# B&R Automation Studio project Tmp_Explorer_V1 (part 2)

#### Main.st - not listed in the package file held
```iecst
// ----------------------------------------------------------------------------------------
//	Function:	mappView explorer
//  Version:	1.08
//	Changed:	03.05.2021
// ----------------------------------------------------------------------------------------

PROGRAM _INIT
	// ----------------------------------------------------------------------------------------
	// Copy pre-configured devices into list
	brsmemcpy(ADR(EXPL.PAR[0].device_list), ADR(EXPL_DEVICE_LIST), SIZEOF(EXPL_DEVICE_LIST));
	brsmemcpy(ADR(EXPL.PAR[1].device_list), ADR(EXPL_DEVICE_LIST), SIZEOF(EXPL_DEVICE_LIST));
	brsstrcpy(ADR(EXPL.PAR[0].device_active), ADR(EXPL.PAR[0].device_list[0]));
	brsstrcpy(ADR(EXPL.PAR[1].device_active), ADR(EXPL.PAR[1].device_list[0]));

	// ----------------------------------------------------------------------------------------
	// Allocate memory for file upload and download
	AsMemPartCreate_0.enable	:= TRUE;
	AsMemPartCreate_0.len		:= EXPL_UPLOAD_DOWNLOAD_SIZE;
	AsMemPartCreate_0();
	IF AsMemPartCreate_0.status <> 0 THEN
		step := CreateError(ERR_MEM_ALLOC, side, step, 'file upload and download alloc failed', ADR(EXPL));
	ELSE
		AsMemPartAllocClear_0.enable	:= TRUE;
		AsMemPartAllocClear_0.ident		:= AsMemPartCreate_0.ident;
		AsMemPartAllocClear_0.len		:= EXPL_UPLOAD_DOWNLOAD_SIZE;
		AsMemPartAllocClear_0();
		IF AsMemPartCreate_0.status <> 0 THEN
			step := CreateError(ERR_MEM_ALLOC, side, step, 'file upload and download clear failed', ADR(EXPL));
		END_IF
	END_IF

	// ----------------------------------------------------------------------------------------
	// Generate HTML messages for web upload
	upload_response[0]	:= '<html><body><form action="/uploadA.html" name="form_upload" method="post" enctype="multipart/form-data" >
	<label for="file-upload" style="font-weight:bold;font-family: sans-serif;font-size:16px;padding:10px 10px;10px;10px;" class="custom-file-upload">Upload</label>
	<input type="file" id="file-upload" style="display:none;" onchange="form.submit()" name="file_selected" content-type="application/octet-stream" />
	</form><body></html> ';
	WebServiceUpload[0].pServiceName := ADR('uploadA.html');
	upload_response[1]	:= '<html><body><form action="/uploadB.html" name="form_upload" method="post" enctype="multipart/form-data" >
	<label for="file-upload" style="font-weight:bold;font-family: sans-serif;font-size:16px;padding:10px 10px;10px;10px;" class="custom-file-upload">Upload</label>
	<input type="file" id="file-upload" style="display:none;" onchange="form.submit()" name="file_selected" content-type="application/octet-stream" />
	</form><body></html> ';
	WebServiceUpload[1].pServiceName := ADR('uploadB.html');

	// ----------------------------------------------------------------------------------------
	// Connect to user device for temporary files used with download all
	REPEAT
		DevLink_0.enable := 1;
		DevLink_0.pDevice := ADR('TMP_USER');
		DevLink_0.pParam := ADR('/DEVICE=F:');
		DevLink_0;
		UNTIL DevLink_0.status <> ERR_FUB_BUSY
	END_REPEAT;
END_PROGRAM

PROGRAM _CYCLIC
	// ----------------------------------------------------------------------------------------
	// Web service driver for file upload
	WebServiceUpload[side].enable 			:= TRUE;
	WebServiceUpload[side].option 			:= httpOPTION_HTTP_11 + httpOPTION_SERVICE_TYPE_NAME;
	WebServiceUpload[side].pRequestData  	:= AsMemPartAllocClear_0.mem;
	WebServiceUpload[side].requestDataSize 	:= EXPL_UPLOAD_DOWNLOAD_SIZE;
	WebServiceUpload[side].pResponseData 	:= ADR(upload_response[side]);
	WebServiceUpload[side].responseDataLen 	:= brsstrlen(ADR(upload_response[side]));
	WebServiceUpload[side]();

	// Reset send command
	IF(WebServiceUpload[side].send = TRUE)  THEN
		WebServiceUpload[side].send := FALSE;
	// Send response when page is loaded or data is posted
	ELSIF(WebServiceUpload[side].status = ERR_OK AND WebServiceUpload[side].send = FALSE) THEN
		WebServiceUpload[side].send := TRUE;
	// New upload data arrived
	ELSIF(WebServiceUpload[side].send = FALSE AND WebServiceUpload[side].requestDataLen > 0 AND EXPL.CMD[side].upload = FALSE) THEN
		// Add delay so that upload can finish
		upload_delay.PT := WebServiceUpload[side].requestDataLen/100000*5;
		upload_delay.IN := TRUE;
		upload_delay();
	END_IF
	// Check new uploaded data
	IF(upload_delay.Q AND EXPL.CMD[side].upload = FALSE) THEN
		upload_delay.IN := FALSE;
		upload_delay();
		EXPL.CMD[side].upload := TRUE;
	END_IF

	// ------------------------------------------------------------------------------------------------
	// Set switches for HMI, these buttons are enabled if there is at least one file or directory
	IF(EXPL.DAT[side].item_num > 0) THEN
		EXPL.VIS[side].enable_button_set_1 := TRUE;
	ELSE
		EXPL.VIS[side].enable_button_set_1 := FALSE;
	END_IF

	// ------------------------------------------------------------------------------------------------
	// Generate device name list for drop down box
	brsmemset(ADR(EXPL.VIS[side].device_list), 0, SIZEOF(EXPL.VIS[side].device_list));
	FOR lx := 0 TO SIZEOF(EXPL.VIS[side].device_list)/SIZEOF(EXPL.VIS[side].device_list[0]) - 1 DO
		IF (EXPL.PAR[side].device_list[lx] <> '') THEN
			String2DataProvider(ADR(EXPL.PAR[side].device_list[lx]), ADR(EXPL.VIS[side].device_list[lx]));
		END_IF
	END_FOR;

	// ------------------------------------------------------------------------------------------------
	// Handle double click for directory change and file view
	IF(EXPL.VIS[side].double_click_event > 0) THEN
		double_click_timer.PT := 50;
		double_click_timer.IN := TRUE;
		double_click_timer();
		IF(EXPL.VIS[side].double_click_event > 1) THEN
			double_click_timer.IN := FALSE;
			double_click_timer();
			EXPL.VIS[side].double_click_event := 0;
			IF(brsmemcmp(ADR(EXPL.DAT[side].item_list[EXPL.VIS[side].item_selected]), ADR('(DIR)'), 5) = 0 OR EXPL.DAT[side].item_list[EXPL.VIS[side].item_selected] = '..') THEN
				EXPL.CMD[side].dir_change := TRUE;
			ELSE
				EXPL.CMD[side].view_file := TRUE;
			END_IF
		END_IF
	END_IF
	IF(double_click_timer.Q) THEN
		double_click_timer.IN := FALSE;
		double_click_timer();
		IF(EXPL.VIS[side].double_click_event > 0) THEN
			EXPL.VIS[side].double_click_event := EXPL.VIS[side].double_click_event - 1;
		END_IF
	END_IF

	//--------------------------------------------------------------------------------------------------
	// Check if parameters are valid
	IF (EXPL.PAR[side].device_active = '') THEN
		step := CreateError(ERR_DEVICE_UNDEFINED, side, step, 'device is not defined', ADR(EXPL));
		RETURN;
	END_IF
	IF (brsstrlen(ADR(EXPL.PAR[side].dir_path)) >= EXPL_DIR_PATH_LENGTH) THEN
		step := CreateError(ERR_PATH_CRITICAL, side, step, 'directory path critical error', ADR(EXPL));
		RETURN;
	END_IF

	// ------------------------------------------------------------------------------------------------
	// Track filter change
	IF (FILTER_AUTO_REFRESH AND brsstrcmp(ADR(old_filter[side]), ADR(EXPL.PAR[side].item_filter)) <> 0) THEN
		brsstrcpy(ADR(old_filter[side]), ADR(EXPL.PAR[side].item_filter));
		EXPL.CMD[side].refresh	:= TRUE;
	END_IF

	// ------------------------------------------------------------------------------------------------
	// Track device name change
	IF(device_active_old[side] <> EXPL.PAR[side].device_active) THEN
		EXPL.PAR[side].dir_path := '';
		EXPL.CMD[side].refresh	:= TRUE;
	END_IF
	device_active_old[side] := EXPL.PAR[side].device_active;

	// ------------------------------------------------------------------------------------------------
	// Stop here if no command is set
	IF (EXPL.CMD[side].refresh = FALSE AND EXPL.CMD[side].dir_change = FALSE AND EXPL.CMD[side].dir_create = FALSE AND EXPL.CMD[side].copy = FALSE AND EXPL.CMD[side].copy_all = FALSE AND EXPL.CMD[side].delete = FALSE AND EXPL.CMD[side].rename = FALSE AND EXPL.CMD[side].view_file = FALSE AND EXPL.CMD[side].download = FALSE AND EXPL.CMD[side].upload = FALSE) THEN
		// --------------------------------------------------------------------------------------------
		// Show current state
		EXPL.status_text := 'Waiting...';
		// --------------------------------------------------------------------------------------------
		// If selection is out of range set it to maximum
		IF ((EXPL.VIS[side].item_selected > EXPL.DAT[side].item_num - 1) AND (EXPL.DAT[side].item_num <> 0)) THEN
			EXPL.VIS[side].item_selected := EXPL.DAT[side].item_num - 1;
		END_IF
		side := NOT side;
		// Enable buttons when command is active
		EXPL.VIS[0].enable_button_set_2 := TRUE;
		EXPL.VIS[1].enable_button_set_2 := TRUE;
		// Reset busy status
		IF(EXPL.ERR.state = 0) THEN
			EXPL.status_no := 0;
		END_IF
		RETURN;
	END_IF

	// Disable buttons when command is active
	EXPL.VIS[0].enable_button_set_1 := FALSE;
	EXPL.VIS[1].enable_button_set_1 := FALSE;
	EXPL.VIS[0].enable_button_set_2 := FALSE;
	EXPL.VIS[1].enable_button_set_2 := FALSE;

	// Clear errors on new command
	brsmemset(ADR(EXPL.ERR), 0, SIZEOF(EXPL.ERR));

	//**************************************************************************************************
	// Cyclic Part
	//**************************************************************************************************
	CASE step OF
		//**********************************************************************************************
		// Wait for command
		//**********************************************************************************************
		EXP_WAIT:
			// ----------------------------------------------------------------------------------------
			// Refresh direcrory information
			IF (EXPL.CMD[side].refresh = TRUE) THEN
				step := EXP_READ_DIR;
			END_IF
			// ----------------------------------------------------------------------------------------
			// Change active directory
			IF (EXPL.CMD[side].dir_change = TRUE) THEN
				// ------------------------------------------------------------------------------------
				// Check if directory name is empty
				IF (EXPL.DAT[side].item_list[EXPL.VIS[side].item_selected] = '') THEN
					step := CreateError(ERR_EMPTY_ITEM, side, step, 'directory name is empty', ADR(EXPL));
				// Check if directory name is valid
				ELSIF((brsmemcmp(ADR(EXPL.DAT[side].item_list[EXPL.VIS[side].item_selected]), ADR('(DIR)'), 5) <> 0) AND (EXPL.DAT[side].item_list[EXPL.VIS[side].item_selected] <> '..'))  THEN
					step := CreateError(ERR_INVALID_ITEM_NAME, side, step, 'this is not a valid directory name', ADR(EXPL));
				// Check if new directory name fits into string
				ELSIF(brsstrlen(ADR(EXPL.DAT[side].item_list[EXPL.VIS[side].item_selected])) - 5 + brsstrlen(ADR(EXPL.PAR[side].dir_path)) + 1 >= EXPL_DIR_PATH_LENGTH) THEN
					step := CreateError(ERR_PATH_EXCEEDS_MAX, side, step, 'directory path exceeds maximum length', ADR(EXPL));
				ELSE
					step := EXP_DIR_CHANGE;
				END_IF
			END_IF
			// ----------------------------------------------------------------------------------------
			// Create a new directory
			IF (EXPL.CMD[side].dir_create = TRUE) THEN
				// ------------------------------------------------------------------------------------
				// Check if new directory name is empty
				IF (EXPL.PAR[side].new_name = '') THEN
					step := CreateError(ERR_EMPTY_ITEM, side, step, 'directory name is empty', ADR(EXPL));
				// Check if new directory name fits into path string
				ELSIF(brsstrlen(ADR(EXPL.PAR[side].new_name)) + brsstrlen(ADR(EXPL.PAR[side].dir_path)) + 1 >= EXPL_DIR_PATH_LENGTH) THEN
					step := CreateError(ERR_PATH_EXCEEDS_MAX, side, step, 'directory path name exceeds maximum length', ADR(EXPL));
				// Check if new directory name fits into directory name string
				ELSIF(brsstrlen(ADR(EXPL.PAR[side].new_name)) + 5 >= EXPL_ITEM_LENGTH) THEN
					step := CreateError(ERR_DIR_EXCEEDS_MAX, side, step, 'directory name exceeds maximum length', ADR(EXPL));
				ELSE
					step := EXP_DIR_CREATE;
				END_IF
			END_IF
			// ----------------------------------------------------------------------------------------
			// Copy one file
			IF (EXPL.CMD[side].copy = TRUE) THEN
				// ------------------------------------------------------------------------------------
				// Make sure that user chooses a valid item
				IF (EXPL.DAT[side].item_list[EXPL.VIS[side].item_selected] = '..') THEN
					step := CreateError(ERR_INVALID_ITEM_NAME, side, step, 'this is not a valid item name', ADR(EXPL));
				ELSE
					item_name := EXPL.DAT[side].item_list[EXPL.VIS[side].item_selected];
					step := EXP_OVERWRITE_1;
				END_IF
			END_IF
			// ----------------------------------------------------------------------------------------
			// Copy all files and folders in this directory
			IF (EXPL.CMD[side].copy_all = TRUE) THEN
				step := EXP_COPY_ALL;
			END_IF
			// ----------------------------------------------------------------------------------------
			// View selected file
			IF (EXPL.CMD[side].view_file = TRUE) THEN
				step := EXP_FILE_VIEW;
			END_IF
			// ----------------------------------------------------------------------------------------
			// Download selected file or directory
			IF (EXPL.CMD[side].download = TRUE) THEN
				EXPL.VIS[side].download_file_url := '';
				item_name := EXPL.DAT[side].item_list[EXPL.VIS[side].item_selected];
				// Make sure selected entry is valid
				IF(brsmemcmp(ADR(item_name), ADR('..'), 2) <> 0) THEN
					// Check if selected item is a single file
					IF(brsmemcmp(ADR(item_name), ADR('(DIR)'), 5) <> 0) THEN
						device_active := EXPL.PAR[side].device_active;
						dir_path := EXPL.PAR[side].dir_path;
						step := EXP_FILE_DOWNLOAD;
					// Selected item is a directory
					ELSE
						ReplaceString(ADR(item_name), ADR('(DIR)'), ADR(''), TRUE);
						step := EXP_FILE_DOWNLOAD_DIR;
					END_IF
				ELSE
					step := CreateError(ERR_DIR_DOWNLOAD_INVALID, side, step, 'item is not a valid directory', ADR(EXPL));
				END_IF
			END_IF
			// ----------------------------------------------------------------------------------------
			// Upload a new file
			IF (EXPL.CMD[side].upload = TRUE) THEN
				step := EXP_FILE_UPLOAD;
			END_IF
			// ----------------------------------------------------------------------------------------
			// Delete the selected file
			IF (EXPL.CMD[side].delete = 1) THEN
				// Check if directory name is empty
				IF (EXPL.DAT[side].item_list[EXPL.VIS[side].item_selected] = '')	THEN
					step := CreateError(ERR_EMPTY_ITEM, side, step, 'item name is empty', ADR(EXPL));
					// Check if new directory name fits into string
				ELSIF(brsstrlen(ADR(EXPL.DAT[side].item_list[EXPL.VIS[side].item_selected])) + brsstrlen(ADR(EXPL.PAR[side].dir_path)) + 1 >= EXPL_DIR_PATH_LENGTH + EXPL_ITEM_LENGTH) THEN
					step := CreateError(ERR_PATH_EXCEEDS_MAX, side, step, 'directory path exceeds maximum length', ADR(EXPL));
					// Make sure that a valid item was selected
				ELSIF(EXPL.DAT[side].item_list[EXPL.VIS[side].item_selected] = '..') THEN
					step := CreateError(ERR_INVALID_ITEM_NAME, side, step, 'this is not a valid item name', ADR(EXPL));
					// Delete a directory
				ELSIF(brsmemcmp(ADR(EXPL.DAT[side].item_list[EXPL.VIS[side].item_selected]), ADR('(DIR)'), 5) = 0)	THEN
					item_name := EXPL.DAT[side].item_list[EXPL.VIS[side].item_selected];
					step := EXP_DIR_DELETE;
				// Delete a file
				ELSE
					item_name := EXPL.DAT[side].item_list[EXPL.VIS[side].item_selected];
					step := EXP_FILE_DELETE;
				END_IF
			END_IF
			// ----------------------------------------------------------------------------------------
			// Rename file or directory
			IF (EXPL.CMD[side].rename = TRUE) THEN
				// ------------------------------------------------------------------------------------
				// Check if new directory name is empty
				IF (EXPL.PAR[side].new_name = '') THEN
					step := CreateError(ERR_EMPTY_ITEM, side, step, 'new name is empty', ADR(EXPL));
				// Make sure that a valid item was selected
				ELSIF (EXPL.DAT[side].item_list[EXPL.VIS[side].item_selected] = '..') THEN
					step := CreateError(ERR_INVALID_ITEM_NAME, side, step, 'this is not a valid item name', ADR(EXPL));
				// Rename a directory
				ELSIF(brsmemcmp(ADR(EXPL.DAT[side].item_list[EXPL.VIS[side].item_selected]), ADR('(DIR)'), 5) = 0)	THEN
					step := EXP_DIR_RENAME;
				// Rename a file
				ELSE
					step := EXP_FILE_RENAME;
				END_IF
			END_IF

			// Set status
			EXPL.status_no := ERR_FUB_BUSY;

		//**********************************************************************************************
		// Read directory information
		//**********************************************************************************************
		EXP_READ_DIR:
			// Show current state
			animation := animation := WorkingStatus(ADR(EXPL), ADR('reading directory...'), animation);
			// ----------------------------------------------------------------------------------------
			// Clear all entrys
			brsmemset(ADR(EXPL.DAT[side]), 0, SIZEOF(EXPL.DAT[side]));
			EXPL.VIS[side].item_selected := 0;
			EXPL.DAT[side].item_num := 0;
			// ----------------------------------------------------------------------------------------
			// Add .. for directory up
			IF(EXPL.PAR[side].dir_path <> '/' AND EXPL.PAR[side].dir_path <> '') THEN
				EXPL.DAT[side].item_list[0] := '..';
				EXPL.DAT[side].item_num := 1;
			END_IF
			// ----------------------------------------------------------------------------------------
			// Set parameters and get device dir
			DInfo.enable 	:= TRUE;
			DInfo.pDevice	:= ADR(EXPL.PAR[side].device_active);
			DInfo.pPath 	:= ADR(EXPL.PAR[side].dir_path);
			DInfo();

			// ----------------------------------------------------------------------------------------
			// OK
			IF (DInfo.status = OK) THEN
				step := EXP_READ_DIR_1;
			// ----------------------------------------------------------------------------------------
			// Device is not available
			ELSIF (DInfo.status = fiERR_FILE_DEVICE) THEN
			 	EXPL.DAT[side].item_list[0] := 'not connected';
				step := CreateError(DInfo.status, side, step, 'not connected', ADR(EXPL));
			// ----------------------------------------------------------------------------------------
			// Device is not available
			ELSIF (DInfo.status = fiERR_DEVICE_MANAGER) THEN
				EXPL.DAT[side].item_list[0] := 'not connected';
				step := CreateError(DInfo.status, side, step, 'check device name and path', ADR(EXPL));
			// Error
			ELSIF (DInfo.status <> ERR_FUB_BUSY) THEN
				step := CreateError(DInfo.status, side, step, 'error dir info', ADR(EXPL));
			END_IF
		//**********************************************************************************************
		// Open directory
		//**********************************************************************************************
		EXP_READ_DIR_1:
			// Add current directory
			IF(EXPL.PAR[side].dir_path = '') THEN
				EXPL.PAR[side].dir_path := '/';
			END_IF
			DOpen.enable 	:= TRUE;
			DOpen.pDevice	:= ADR(EXPL.PAR[side].device_active);
			DOpen.pName 	:= ADR(EXPL.PAR[side].dir_path);
			DOpen();

			// ----------------------------------------------------------------------------------------
			// OK
			IF (DOpen.status = OK) THEN
				has_oversized_items := FALSE;
				step := EXP_READ_DIR_2;
			// Error
			ELSIF (DOpen.status <> ERR_FUB_BUSY) THEN
				step := CreateError(DOpen.status, side, step, 'error dir open', ADR(EXPL));
			END_IF;
		//**********************************************************************************************
		// Read file directory information
		//**********************************************************************************************
	 	EXP_READ_DIR_2:
			DRead.enable 	:= TRUE;
			DRead.ident		:= DOpen.ident;
			DRead.pData 	:= ADR(lDirReadData);
			DRead.data_len 	:= SIZEOF(lDirReadData);
			DRead();

			// ----------------------------------------------------------------------------------------
			// OK
			IF (DRead.status = OK) THEN
				// ------------------------------------------------------------------------------------
				// Verify that we still have space in list
				IF (EXPL.DAT[side].item_num < SIZEOF(EXPL.DAT[side].item_list)/SIZEOF(EXPL.DAT[side].item_list[0])) THEN
					// --------------------------------------------------------------------------------
					// Make sure file name contains filter
					IF (brsstrlen(ADR(EXPL.PAR[side].item_filter)) = 0 OR IsInstr(ADR(lDirReadData.Filename), ADR(EXPL.PAR[side].item_filter))) THEN
						brsmemset(ADR(tmp_str1), 0, SIZEOF(tmp_str1));
						// ----------------------------------------------------------------------------
						// Read file information
						IF (lDirReadData.Mode = fiFILE) THEN
							IF (brsstrlen(ADR(lDirReadData.Filename)) < EXPL_ITEM_LENGTH) THEN
								brsstrcpy(ADR(tmp_str1), ADR(lDirReadData.Filename));
								// --------------------------------------------------------------------
								// Generate file size
								IF (lDirReadData.Filelength > 1048576) THEN
									brsitoa(lDirReadData.Filelength/1048576, ADR(tmp_str2));
									brsstrcat(ADR(tmp_str2), ADR('M'));
								ELSIF (lDirReadData.Filelength > 1024) THEN
									brsitoa(lDirReadData.Filelength/1024, ADR(tmp_str2));
									brsstrcat(ADR(tmp_str2), ADR('K'));
								ELSE
									brsitoa(lDirReadData.Filelength, ADR(tmp_str2));
								END_IF
								InsertRecName(ADR(EXPL), tmp_str1, tmp_str2, side);
								EXPL.DAT[side].item_num := EXPL.DAT[side].item_num + 1;
							ELSE
								has_oversized_items := TRUE;
							END_IF
						// ----------------------------------------------------------------------------
						// Read directory information
						ELSIF (brsstrcmp(ADR(lDirReadData.Filename), ADR('.')) <> 0 AND brsstrcmp(ADR(lDirReadData.Filename), ADR('..')) <> 0 AND brsstrcmp(ADR(lDirReadData.Filename), ADR('System Volume Information')) <> 0) THEN
							IF (brsstrlen(ADR(lDirReadData.Filename)) < EXPL_ITEM_LENGTH-5) THEN
								// Copy directory name
								tmp_str1 := '(DIR)';
								brsstrcat(ADR(tmp_str1), ADR(lDirReadData.Filename));
								InsertRecName(ADR(EXPL), tmp_str1, '', side);
								EXPL.DAT[side].item_num := EXPL.DAT[side].item_num + 1;
							ELSE
								has_oversized_items := TRUE;
							END_IF
						END_IF
					END_IF
				ELSE
					step := CreateError(ERR_MAX_FILES_REACHED, side, step, 'maximum number of files reached', ADR(EXPL));
				END_IF
			// Last entry reached
			ELSIF (DRead.status = fiERR_NO_MORE_ENTRIES) THEN
				step := EXP_READ_DIR_3;
			// Error
			ELSIF (DRead.status <> ERR_FUB_BUSY) THEN
				step := CreateError(DRead.status, side, step, 'error dir read', ADR(EXPL));
			END_IF
		//**********************************************************************************************
		// Close directory information
		//**********************************************************************************************
		EXP_READ_DIR_3:
			DClose.enable 	:= TRUE;
			DClose.ident	:= DOpen.ident;
			DClose();

			// ----------------------------------------------------------------------------------------
			// OK
			IF (DClose.status = OK) THEN
				// Report error from dir read
				IF (DRead.status <> ERR_OK AND DRead.status <> fiERR_NO_MORE_ENTRIES) THEN
					step := CreateError(DRead.status, side, step, 'error dir read', ADR(EXPL));
				ELSE
					DClose.ident := 0;
					step := EXP_READ_DIR_4;
				END_IF
			// Error
			ELSIF (DClose.status <> ERR_FUB_BUSY) THEN
				step := CreateError(DClose.status, side, step, 'error dir close', ADR(EXPL));
			END_IF
		//**********************************************************************************************
		// Get device memory information
		//**********************************************************************************************
		EXP_READ_DIR_4:
			DMemInfo.enable 	:= TRUE;
			DMemInfo.pDevice	:= ADR(EXPL.PAR[side].device_active);
			DMemInfo();

			// ----------------------------------------------------------------------------------------
			// OK
			IF (DMemInfo.status = OK) THEN
				// Transfer device memory information
				EXPL.DAT[side].device_free := UDINT_TO_INT(DMemInfo.freemem/1048576);
				EXPL.DAT[side].device_size := UDINT_TO_INT(DMemInfo.memsize/1048576);
				// Select item after copy->refresh
				IF(do_select <> 0) THEN
					FOR ly:=0 TO EXPL.DAT[NOT USINT_TO_BOOL(do_select-1)].item_num DO
						IF(EXPL.DAT[USINT_TO_BOOL(do_select-1)].item_list[EXPL.VIS[USINT_TO_BOOL(do_select-1)].item_selected] = EXPL.DAT[NOT USINT_TO_BOOL(do_select-1)].item_list[ly]) THEN
							EXIT;
						END_IF
					END_FOR;
					EXPL.VIS[NOT USINT_TO_BOOL(do_select-1)].item_selected := ly;
					do_select := 0;
				END_IF
				// Reset command and return to wait state
				EXPL.CMD[side].refresh	:= FALSE;
				IF(has_oversized_items) THEN
					step := CreateError(ERR_NAME_EXCEEDS_MAX, side, step, 'one or more names exceeds maximum length', ADR(EXPL));
				ELSE
					step := EXP_WAIT;
				END_IF
				// Error
			ELSIF (DMemInfo.status <> ERR_FUB_BUSY) THEN
				step := CreateError(DMemInfo.status, side, step, 'error reading device memory information', ADR(EXPL));
			END_IF
		//**********************************************************************************************
		// Change directory
		//**********************************************************************************************
		EXP_DIR_CHANGE:
			// ----------------------------------------------------------------------------------------
			// Move one directory up
			IF (EXPL.DAT[side].item_list[EXPL.VIS[side].item_selected] = '..') THEN
				lx := brsstrlen(ADR(EXPL.PAR[side].dir_path));
				WHILE lx>0 DO
					IF(brsmemcmp(ADR(EXPL.PAR[side].dir_path) + lx, ADR('/'), 1) = 0) THEN
						EXIT;
					ELSE
						brsmemset(ADR(EXPL.PAR[side].dir_path) + lx, 0, 1);
					END_IF
					lx := lx -1;
				END_WHILE
				brsmemset(ADR(EXPL.PAR[side].dir_path) + lx, 0, 1);
			// ----------------------------------------------------------------------------------------
			// Move one directory down
			ELSE
				// Add slash if not in root
				IF(EXPL.PAR[side].dir_path <> '/') THEN
					brsstrcat(ADR(EXPL.PAR[side].dir_path), ADR('/'));
				END_IF
				brsstrcat(ADR(EXPL.PAR[side].dir_path), ADR(EXPL.DAT[side].item_list[EXPL.VIS[side].item_selected]) + 5);
				EXPL.CMD[side].refresh := 1;
			END_IF
			// Reset command and return to wait state
			EXPL.VIS[side].item_selected	:= 0;
			EXPL.CMD[side].dir_change 		:= 0;
			EXPL.CMD[side].refresh 			:= TRUE;
			step							:= EXP_WAIT;
		//**********************************************************************************************
		// Copy all items
		//**********************************************************************************************
		EXP_COPY_ALL:
			// Show current state
			animation := animation := WorkingStatus(ADR(EXPL), ADR('copying files and folders...'), animation);

			EXPL.VIS[side].item_selected := 0;
			// ----------------------------------------------------------------------------------------
			// Skip dots at the beginning of the list
			IF (EXPL.DAT[side].item_list[EXPL.VIS[side].item_selected] = '..') THEN
				EXPL.VIS[side].item_selected := EXPL.VIS[side].item_selected + 1;
			END_IF
			// Check first entry
			IF(brsmemcmp(ADR(EXPL.DAT[side].item_list[EXPL.VIS[side].item_selected]), ADR('(DIR)'), 5) = 0) THEN
				step := EXP_DIR_COPY;
			ELSE
				step := EXP_FILE_COPY;
			END_IF
		//**********************************************************************************************
		// Copy files
		//**********************************************************************************************
		EXP_FILE_COPY:
			// Show current state
			animation := WorkingStatus(ADR(EXPL), ADR('copying file...'), animation);

			// -----------------------------------------------------------------.----------------------
			// Proceed with copy all until last file is copied
			IF ((EXPL.VIS[side].item_selected < SIZEOF(EXPL.DAT[side].item_list)/SIZEOF(EXPL.DAT[side].item_list[0])) AND (EXPL.VIS[side].item_selected < EXPL.DAT[side].item_num)) THEN
				// ------------------------------------------------------------------------------------
				// Check if file name is empty
				IF (EXPL.DAT[side].item_list[EXPL.VIS[side].item_selected] <> '') THEN
					// --------------------------------------------------------------------------------
					// Check if new file name fits into string
					IF(brsstrlen(ADR(EXPL.DAT[side].item_list[EXPL.VIS[side].item_selected])) < EXPL_ITEM_LENGTH) THEN
						// ----------------------------------------------------------------------------
						// Initialize copy structure
						CreateCompletePath(EXPL.PAR[side].dir_path, EXPL.DAT[side].item_list[EXPL.VIS[side].item_selected], ADR(tmp_str3));
						CreateCompletePath(EXPL.PAR[NOT side].dir_path, EXPL.DAT[side].item_list[EXPL.VIS[side].item_selected], ADR(tmp_str4));
						FCopy.enable 	:= 1;
						FCopy.pSrcDev	:= ADR(EXPL.PAR[side].device_active);
						FCopy.pSrc		:= ADR(tmp_str3);
						FCopy.pDestDev  := ADR(EXPL.PAR[NOT side].device_active);
						FCopy.pDest		:= ADR(tmp_str4);
						FCopy.option 	:= FILE_OW_DETMEM;
						FCopy();

						// ----------------------------------------------------------------------------
						// OK
						IF (FCopy.status = OK AND EXPL.CMD[side].copy = 1) THEN
							// Select entry, reset command and refresh directory
							IF(COPY_AUTO_REFRESH = TRUE) THEN
								EXPL.CMD[NOT side].refresh := TRUE;
							END_IF
							IF(COPY_AUTO_SELECT = TRUE) THEN
								do_select := BOOL_TO_USINT(side) + 1;
							END_IF
							EXPL.CMD[side].copy	:= FALSE;
							step := EXP_WAIT;
						// ----------------------------------------------------------------------------
						// Proceed with next file
						ELSIF (FCopy.status = OK) THEN
							EXPL.VIS[side].item_selected := EXPL.VIS[side].item_selected + 1;
						ELSIF (FCopy.status <> ERR_FUB_BUSY) THEN
							step := CreateError(FCopy.status, side, step, 'error copying file', ADR(EXPL));
						END_IF
					// File name is too long
					ELSE
						step := CreateError(ERR_NAME_EXCEEDS_MAX, side, step, 'file name exceeds maximum length', ADR(EXPL));
					END_IF
				// File name  is empty
				ELSE
					step := CreateError(ERR_EMPTY_ITEM, side, step, 'file name is empty', ADR(EXPL));
				END_IF
			// ----------------------------------------------------------------------------------------
			// Finish copy all
			ELSE
				// Reset command and refresh directory
				IF(COPY_AUTO_REFRESH = TRUE) THEN
					EXPL.CMD[NOT side].refresh := TRUE;
				END_IF
				EXPL.CMD[side].copy_all			:= FALSE;
				EXPL.VIS[side].item_selected 	:= 0;
				step							:= EXP_WAIT;
			END_IF
		//**********************************************************************************************
		// Copy directory
		//**********************************************************************************************
		EXP_DIR_COPY:
			// Show current state
			animation := WorkingStatus(ADR(EXPL), ADR('copying directory...'), animation);

			// ----------------------------------------------------------------------------------------
			// Proceed with copy all until last file is copied
			IF ((EXPL.VIS[side].item_selected < SIZEOF(EXPL.DAT[side].item_list)/SIZEOF(EXPL.DAT[side].item_list[0])) AND (EXPL.VIS[side].item_selected < EXPL.DAT[side].item_num)) THEN
				IF (EXPL.DAT[side].item_list[EXPL.VIS[side].item_selected] <> '') THEN
					// --------------------------------------------------------------------------------
					// Check if new directory name fits into path string
					IF(brsstrlen(ADR(EXPL.DAT[side].item_list[EXPL.VIS[side].item_selected])) + brsstrlen(ADR(EXPL.PAR[NOT side].dir_path)) + 1 < EXPL_DIR_PATH_LENGTH) THEN
						// ----------------------------------------------------------------------------
						// Initialize copy structure
						CreateCompletePath(EXPL.PAR[side].dir_path, EXPL.DAT[side].item_list[EXPL.VIS[side].item_selected], ADR(tmp_str3));
						CreateCompletePath(EXPL.PAR[NOT side].dir_path, EXPL.DAT[side].item_list[EXPL.VIS[side].item_selected], ADR(tmp_str4));
						// ----------------------------------------------------------------------------
						// Make sure we are not copying directories recursively
						IF((EXPL.PAR[side].device_active = EXPL.PAR[NOT side].device_active) AND ((brsmemcmp(ADR(tmp_str3), ADR(tmp_str4), brsstrlen(ADR(tmp_str3))) = 0) OR (brsmemcmp(ADR(tmp_str4), ADR(tmp_str3), brsstrlen(ADR(tmp_str4))) = 0))) THEN
							step := CreateError(ERR_PATH_RECURSIVE, side, step, 'can not copy directory into itself', ADR(EXPL));
						ELSE
							DCopy.enable 	:= 1;
							DCopy.pSrcDev	:= ADR(EXPL.PAR[side].device_active);
							DCopy.pSrcDir	:= ADR(tmp_str3);
							DCopy.pDestDev 	:= ADR(EXPL.PAR[NOT side].device_active);
							DCopy.pDestDir 	:= ADR(tmp_str4);
							DCopy.option 	:= fiOVERWRITE;
							DCopy();

							// ----------------------------------------------------------------------------
							// OK
							IF (DCopy.status = OK AND EXPL.CMD[side].copy = 1) THEN
								// Reset command and refresh directory
								IF(COPY_AUTO_REFRESH = TRUE) THEN
									EXPL.CMD[NOT side].refresh := TRUE;
								END_IF
								IF (COPY_AUTO_SELECT = TRUE) THEN
									do_select := BOOL_TO_USINT(side) + 1;
								END_IF
								EXPL.CMD[side].copy	:= FALSE;
								step := EXP_WAIT;
							// ----------------------------------------------------------------------------
							// Proceed with next directory
							ELSIF (DCopy.status = OK) THEN
								EXPL.VIS[side].item_selected := EXPL.VIS[side].item_selected + 1;
								// Switch to file copy when no more directory can be found
								IF(brsmemcmp(ADR(EXPL.DAT[side].item_list[EXPL.VIS[side].item_selected]), ADR('(DIR)'), 5) <> 0) THEN
									step := EXP_FILE_COPY;
								END_IF
							// Error
							ELSIF (DCopy.status <> ERR_FUB_BUSY) THEN
								step := CreateError(DCopy.status, side, step, 'error copying directory', ADR(EXPL));
							END_IF
						END_IF
					// Directory name is too long
					ELSE
						step := CreateError(ERR_PATH_EXCEEDS_MAX, side, step, 'directory path name exceeds maximum length', ADR(EXPL));
					END_IF
				// Directory name is empty
				ELSE
					step := CreateError(ERR_EMPTY_ITEM, side, step, 'directory name is empty', ADR(EXPL));
				END_IF
			// ----------------------------------------------------------------------------------------
			// Finish copy all
			ELSE
				// Reset command and refresh directory
				IF (COPY_AUTO_REFRESH = TRUE) THEN
					EXPL.CMD[NOT side].refresh := TRUE;
				END_IF
				EXPL.CMD[side].copy_all := FALSE;
				EXPL.VIS[side].item_selected := 0;
				step := EXP_WAIT;
			END_IF
		//**********************************************************************************************
		// Delete selected file
		//**********************************************************************************************
		EXP_FILE_DELETE:
			// Show current state
			animation := WorkingStatus(ADR(EXPL), ADR('deleting file...'), animation);

			// ----------------------------------------------------------------------------------------
			// Initialize file delete structure
			CreateCompletePath(EXPL.PAR[side].dir_path, item_name, ADR(tmp_str3));
			FDelete.enable		:= TRUE;
			FDelete.pDevice 	:= ADR(EXPL.PAR[side].device_active);
			FDelete.pName		:= ADR(tmp_str3);
			FDelete();

			// ----------------------------------------------------------------------------------------
			// OK
			IF (FDelete.status = OK) THEN
				// Reset command delete and return to wait state
				IF(EXPL.CMD[side].delete = TRUE) THEN
					EXPL.CMD[side].delete 	:= FALSE;
					EXPL.CMD[side].refresh  := TRUE;
					step := EXP_WAIT;
				// Proceed with command upload
				ELSE
					step := EXP_FILE_UPLOAD_1;
				END_IF
			// Error
			ELSIF (FDelete.status <> ERR_FUB_BUSY) THEN
				step := CreateError(FDelete.status, side, step, 'error deleting file', ADR(EXPL));
			END_IF
		//**********************************************************************************************
		// Rename selected file
		//**********************************************************************************************
		EXP_FILE_RENAME:
			// Show current state
			animation := WorkingStatus(ADR(EXPL), ADR('renaming file...'), animation);

			// ----------------------------------------------------------------------------------------
			// Initialize file delete structure
			CreateCompletePath(EXPL.PAR[side].dir_path, EXPL.DAT[side].item_list[EXPL.VIS[side].item_selected], ADR(tmp_str2));
			CreateCompletePath(EXPL.PAR[side].dir_path, EXPL.PAR[side].new_name, ADR(tmp_str3));
			FRename.enable		:= TRUE;
			FRename.pDevice 	:= ADR(EXPL.PAR[side].device_active);
			FRename.pName		:= ADR(tmp_str2);
			FRename.pNewName	:= ADR(tmp_str3);
			FRename();

			// ----------------------------------------------------------------------------------------
			// OK
			IF (FRename.status = OK) THEN
				// Reset command and return to wait state
				EXPL.CMD[side].rename 	:= FALSE;
				EXPL.CMD[side].refresh  := TRUE;
				step := EXP_WAIT;
				// Error
			ELSIF (FRename.status <> ERR_FUB_BUSY) THEN
				step := CreateError(FRename.status, side, step, 'error renaming file', ADR(EXPL));
			END_IF
		//**********************************************************************************************
		// View selected file
		//**********************************************************************************************
		EXP_FILE_VIEW:
			CreateCompletePath(EXPL.PAR[side].dir_path, EXPL.DAT[side].item_list[EXPL.VIS[side].item_selected], ADR(tmp_str1));

			FOR lx:=0 TO SIZEOF(EXPL_VIEW_FILTER)/SIZEOF(EXPL_VIEW_FILTER[0]) - 1 DO
				IF(brsstrlen(ADR(tmp_str1)) >= brsstrlen(ADR(EXPL_VIEW_FILTER[lx])) AND EXPL_VIEW_FILTER[lx] <> '') THEN
					// --------------------------------------------------------------------------------
					// Verify that file name contains filter
					IF(brsmemcmp(ADR(tmp_str1) + brsstrlen(ADR(tmp_str1)) - brsstrlen(ADR(EXPL_VIEW_FILTER[lx])) , ADR(EXPL_VIEW_FILTER[lx]), brsstrlen(ADR(EXPL_VIEW_FILTER[lx]))) = 0) THEN
						EXPL.VIS[side].view_file_path := '/FileDevice:';
						brsstrcat(ADR(EXPL.VIS[side].view_file_path), ADR(EXPL.PAR[side].device_active));
						brsstrcat(ADR(EXPL.VIS[side].view_file_path), ADR(tmp_str1));
						EXPL.CMD[side].view_file := FALSE;
						EXPL.VIS[side].view_file := TRUE;
						step := EXP_WAIT;
						RETURN;
					END_IF
				END_IF
			END_FOR;
			step := CreateError(FRename.status, side, step, 'error this file extension is not supported for viewing', ADR(EXPL));
		//**********************************************************************************************
		// Download file
		//**********************************************************************************************
		EXP_FILE_DOWNLOAD:
			// ----------------------------------------------------------------------------------------
			// Initialize file open structure
			CreateCompletePath(dir_path, item_name, ADR(tmp_str1));
			FOpen.enable	:= TRUE;
			FOpen.pDevice 	:= ADR(device_active);
			FOpen.pFile		:= ADR(tmp_str1);
			FOpen();

			// ----------------------------------------------------------------------------------------
			// OK
			IF (FOpen.status = OK) THEN
				// Make sure file fits into memory
				IF(FOpen.filelen <= EXPL_UPLOAD_DOWNLOAD_SIZE) THEN
					// Clear memory and reset web service
					brsmemset(AsMemPartAllocClear_0.mem, 0, EXPL_UPLOAD_DOWNLOAD_SIZE);
					WebserviceDownload.enable := FALSE;
					WebserviceDownload();
					step := EXP_FILE_DOWNLOAD_1;
				// File is too large
				ELSE
					tmp_str1 := 'download file exceeds maximum buffer size of ';
					brsitoa(EXPL_UPLOAD_DOWNLOAD_SIZE, ADR(tmp_str2));
					brsstrcat(ADR(tmp_str1), ADR(tmp_str2));
					brsstrcat(ADR(tmp_str1), ADR(' bytes'));
					// Delete old zip file before generating an error
					IF(IsInstr(ADR(item_name), ADR('.tar.gz'))) THEN
						step := EXP_FILE_DOWNLOAD_5;
					ELSE
						step := CreateError(ERR_MEM_DOWNLOAD, side, step, tmp_str1, ADR(EXPL));
					END_IF
				END_IF;
				// Error
			ELSIF (FOpen.status <> ERR_FUB_BUSY) THEN
				step := CreateError(FOpen.status, side, step, 'error opening file for download', ADR(EXPL));
			END_IF
		//**********************************************************************************************
		// Download file
		//**********************************************************************************************
		EXP_FILE_DOWNLOAD_1:
			// ----------------------------------------------------------------------------------------
			// Initialize file read structure
			FRead.enable	:= TRUE;
			FRead.ident		:= FOpen.ident;
			FRead.len		:= FOpen.filelen;
			FRead.pDest		:= AsMemPartAllocClear_0.mem;
			FRead();

			// ----------------------------------------------------------------------------------------
			// OK
			IF (FRead.status = OK) THEN
				step := EXP_FILE_DOWNLOAD_2;
			// Error
			ELSIF (FRead.status <> ERR_FUB_BUSY) THEN
				step := CreateError(FRead.status, side, step, 'error reading file for download', ADR(EXPL));
			END_IF
		//**********************************************************************************************
		// Download file
		//**********************************************************************************************
		EXP_FILE_DOWNLOAD_2:
			// ----------------------------------------------------------------------------------------
			// Initialize file close structure
			FClose.enable	:= TRUE;
			FClose.ident	:= FOpen.ident;
			FClose();

			// ----------------------------------------------------------------------------------------
			// OK
			IF (FClose.status = OK) THEN
				download_timeout.IN := FALSE;
				download_timeout();
				step := EXP_FILE_DOWNLOAD_3;
			// Error
			ELSIF (FClose.status <> ERR_FUB_BUSY) THEN
				step := CreateError(FClose.status, side, step, 'error closing file for download', ADR(EXPL));
			END_IF
		//**********************************************************************************************
		// Download file - web service
		//**********************************************************************************************
		EXP_FILE_DOWNLOAD_3:
			// ----------------------------------------------------------------------------------------
			// Create response header
			response_header_data :=  'Content-Type: application/octet-stream; Content-Transfer-Encoding: binary; Content-Disposition: attachment; filename="';
			brsstrcpy(ADR(tmp_str1), ADR(item_name));
			ReplaceString(ADR(tmp_str1), ADR(' '), ADR('%20'), FALSE);
			brsstrcat(ADR(response_header_data), ADR(tmp_str1));
			brsstrcat(ADR(response_header_data), ADR('"'));

			// ----------------------------------------------------------------------------------------
			// Pre-configure web service for download
			response_header.rawHeader.pData 	:= ADR(response_header_data);
			response_header.rawHeader.dataSize 	:= SIZEOF(response_header_data);
			response_header.rawHeader.dataLen 	:= brsstrlen(ADR(response_header_data));

			// ----------------------------------------------------------------------------------------
			// Start web service
			WebserviceDownload.enable 			:= TRUE;
			WebserviceDownload.option 			:= httpOPTION_HTTP_10 + httpOPTION_SERVICE_TYPE_NAME;
			WebserviceDownload.pResponseData 	:= AsMemPartAllocClear_0.mem;
			WebserviceDownload.pResponseHeader	:= ADR(response_header);
			WebserviceDownload.pServiceName 	:= ADR(tmp_str1);
			WebserviceDownload.responseDataLen 	:= FOpen.filelen;
			WebserviceDownload();

			// ----------------------------------------------------------------------------------------
			// Timeout if file is not pulled from browser
			download_timeout.IN := TRUE;
			download_timeout.PT := 300 + FOpen.filelen/10000;
			download_timeout();
			IF(download_timeout.Q) THEN
				step := CreateError(ERR_TIMEOUT_DOWNLOAD, side, step, 'error download response timed out', ADR(EXPL));
			END_IF

			// ----------------------------------------------------------------------------------------
			// Set URL
			IF (WebserviceDownload.status = ERR_FUB_BUSY AND EXPL.VIS[side].download_file_url = '') THEN
				brsstrcat(ADR(EXPL.VIS[side].download_file_url), ADR(item_name));
			// Start sending data
			ELSIF (WebserviceDownload.status = OK AND WebserviceDownload.send = FALSE AND EXPL.VIS[side].download_file_url <> '') THEN
				WebserviceDownload.send := TRUE;
			// Sending data finished
			ELSIF (WebserviceDownload.send = TRUE) THEN
				step := EXP_FILE_DOWNLOAD_4;
				// Error
			ELSIF (WebserviceDownload.status <> ERR_FUB_BUSY AND WebserviceDownload.status <> OK) THEN
				step := CreateError(WebserviceDownload.status, side, step, 'error sending web response', ADR(EXPL));
			END_IF
		//**********************************************************************************************
		// Download file - web service
		//**********************************************************************************************
		EXP_FILE_DOWNLOAD_4:
			WebserviceDownload();
			download_timeout();
			IF(download_timeout.Q) THEN
				step := CreateError(ERR_TIMEOUT_DOWNLOAD, side, step, 'error download response timed out', ADR(EXPL));
			END_IF

			// ----------------------------------------------------------------------------------------
			// Finish sending data
			IF (WebserviceDownload.phase = httpPHASE_WAITING) THEN
				EXPL.VIS[side].download_file_url := '';
				WebserviceDownload.send := FALSE;
				// Download is a directory
				IF(IsInstr(ADR(item_name), ADR('.tar.gz'))) THEN
					step := EXP_FILE_DOWNLOAD_5;
				// Download is a single file
				ELSE
					EXPL.CMD[side].download	:= FALSE;
					step := EXP_WAIT;
				END_IF
				// Error
			ELSIF (WebserviceDownload.status <> ERR_FUB_BUSY) THEN
				step := CreateError(WebserviceDownload.status, side, step, 'error sending web response', ADR(EXPL));
			END_IF
		//**********************************************************************************************
		// Delete old zip file after download
		//**********************************************************************************************
		EXP_FILE_DOWNLOAD_5:
			// Show current state
			animation := WorkingStatus(ADR(EXPL), ADR('deleting old zip file...'), animation);

			// ----------------------------------------------------------------------------------------
			// Initialize file delete structure
			FDelete.enable		:= TRUE;
			FDelete.pDevice 	:= ADR('TMP_USER');
			FDelete.pName		:= ADR(item_name);
			FDelete();

			// ----------------------------------------------------------------------------------------
			// OK
			IF (FDelete.status = OK) THEN
				// Generate error when file was too large
				IF(FOpen.filelen > EXPL_UPLOAD_DOWNLOAD_SIZE) THEN
					step := CreateError(ERR_MEM_DOWNLOAD, side, step, tmp_str1, ADR(EXPL));
				// Finish directory download
				ELSE
					EXPL.CMD[side].download	:= FALSE;
					step := EXP_WAIT;
				END_IF
			// Error
			ELSIF (FDelete.status <> ERR_FUB_BUSY) THEN
				step := CreateError(FDelete.status, side, step, 'error deleting old zip file', ADR(EXPL));
			END_IF
		//**********************************************************************************************
		// Download all files
		//**********************************************************************************************
		EXP_FILE_DOWNLOAD_DIR:
			// Show current state
			animation := WorkingStatus(ADR(EXPL), ADR('processing directory...'), animation);
			tmp_str1 := item_name;
			brsstrcat(ADR(tmp_str1), ADR('.tar.gz'));

			// ----------------------------------------------------------------------------------------
			// Initialize file zip structure
			CreateCompletePath(EXPL.PAR[side].dir_path, EXPL.DAT[side].item_list[EXPL.VIS[side].item_selected], ADR(tmp_str2));

			zipArchive_0.enable := 1;
			zipArchive_0.pArchiveDevice := ADR('TMP_USER');
			zipArchive_0.pArchiveFile := ADR(tmp_str1);
			zipArchive_0.pSrcDevice := ADR(EXPL.PAR[side].device_active);
			zipArchive_0.pSrcFile := ADR(tmp_str2);
			zipArchive_0.pOptions := ADR('/COMPRESSION_LEVEL=7');
			zipArchive_0();

			// ----------------------------------------------------------------------------------------
			// OK
			IF (zipArchive_0.status = OK) THEN
				item_name := tmp_str1;
				device_active := 'TMP_USER';
				dir_path := '';
				step := EXP_FILE_DOWNLOAD;
			// Error
			ELSIF (zipArchive_0.status <> ERR_FUB_BUSY) THEN
				step := CreateError(zipArchive_0.status, side, step, 'error creating zip file', ADR(EXPL));
			END_IF
		//**********************************************************************************************
		// Upload file - verify parameters
		//**********************************************************************************************
		EXP_FILE_UPLOAD:
			// Show current state
			animation := WorkingStatus(ADR(EXPL), ADR('uploading file...'), animation);

			// Make sure data fits into memory
			IF(WebServiceUpload[side].requestDataLen < EXPL_UPLOAD_DOWNLOAD_SIZE) THEN
				// Find file name start
				file_name_start := FindInMem(AsMemPartAllocClear_0.mem, WebServiceUpload[side].requestDataLen, ADR('filename="'), brsstrlen(ADR('filename="')), FALSE) + brsstrlen(ADR('filename="'));
				IF(file_name_start > 0) THEN
					// Find end of file name
					file_name_len := FindInMem(AsMemPartAllocClear_0.mem+file_name_start, WebServiceUpload[side].requestDataLen-file_name_start, ADR('"$r$n'), brsstrlen(ADR('"$r$n')), FALSE);
					IF(file_name_len > 0) THEN
						// Make sure file name is not too long
						IF(file_name_len <= EXPL_ITEM_LENGTH) THEN
							// Store file name
							brsmemset(ADR(item_name), 0, SIZEOF(item_name));
							brsmemcpy(ADR(item_name), AsMemPartAllocClear_0.mem+file_name_start, file_name_len);
							// Find start of data
							file_data_start := FindInMem(AsMemPartAllocClear_0.mem, WebServiceUpload[side].requestDataLen, ADR('Content-Type:'), brsstrlen(ADR('Content-Type:')), FALSE) + brsstrlen(ADR('Content-Type:'));
							IF(file_data_start > 0) THEN
								// Find end of data
								file_data_start := FindInMem(AsMemPartAllocClear_0.mem+file_data_start, WebServiceUpload[side].requestDataLen-file_data_start, ADR('$r$n$r$n'), brsstrlen(ADR('$r$n$r$n')), FALSE) + brsstrlen(ADR('$r$n$r$n')) + file_data_start;
								file_data_len := FindInMem(AsMemPartAllocClear_0.mem+file_data_start, WebServiceUpload[side].requestDataLen-file_data_start, ADR('$r$n------'), brsstrlen(ADR('$r$n------')), TRUE);
								// When file name and data is correct procceed with saving data to file
								IF(file_data_len > 0) THEN
									step := EXP_OVERWRITE_1;
									RETURN;
								ELSE
									step := CreateError(ERR_SIZE_DATA_UPLOAD, side, step, 'data end not found in upload response', ADR(EXPL));
								END_IF
							// Data start not found in upload response
							ELSE
								step := CreateError(ERR_POS_DATA_UPLOAD, side, step, 'data start not found in upload response', ADR(EXPL));
							END_IF
						// File name is too long in upload response
						ELSE
							step := CreateError(ERR_LEN_NAME_UPLOAD, side, step, 'file name is too long in upload response', ADR(EXPL));
						END_IF
					// File name end not found in upload response
					ELSE
						step := CreateError(ERR_SIZE_NAME_UPLOAD, side, step, 'file name end not found in upload response', ADR(EXPL));
					END_IF
				// File name start not found in upload response
				ELSE
					step := CreateError(ERR_POS_NAME_UPLOAD, side, step, 'file name position not found in upload response', ADR(EXPL));
				END_IF
			// Upload file exceeds maximum buffer size
			ELSE
				tmp_str1 := 'upload file exceeds maximum buffer size of ';
				brsitoa(EXPL_UPLOAD_DOWNLOAD_SIZE, ADR(tmp_str2));
				brsstrcat(ADR(tmp_str1), ADR(tmp_str2));
				brsstrcat(ADR(tmp_str1), ADR(' bytes'));
				step := CreateError(ERR_MEM_UPLOAD, side, step, tmp_str1, ADR(EXPL));
			END_IF
			// Reset upload buffer and function block
			brsmemset(AsMemPartAllocClear_0.mem, 0, EXPL_UPLOAD_DOWNLOAD_SIZE);
			EXPL.VIS[side].reload_upload := TRUE;
			WebServiceUpload[side].enable := FALSE;
			WebServiceUpload[side]();
		//**********************************************************************************************
		// Upload file
		//**********************************************************************************************
		EXP_FILE_UPLOAD_1:
			// ----------------------------------------------------------------------------------------
			// Initialize file create structure
			CreateCompletePath(EXPL.PAR[side].dir_path, item_name, ADR(tmp_str1));
			FCreate.enable	:= TRUE;
			FCreate.pDevice := ADR(EXPL.PAR[side].device_active);
			FCreate.pFile	:= ADR(tmp_str1);
			FCreate();

			// ----------------------------------------------------------------------------------------
			// OK
			IF (FCreate.status = OK) THEN
				step := EXP_FILE_UPLOAD_2;
			// Error
			ELSIF (FCreate.status <> ERR_FUB_BUSY) THEN
				step := CreateError(FCreate.status, side, step, 'error creating file from upload', ADR(EXPL));
				// Reset upload buffer and function block
				brsmemset(AsMemPartAllocClear_0.mem, 0, EXPL_UPLOAD_DOWNLOAD_SIZE);
				EXPL.VIS[side].reload_upload := TRUE;
				WebServiceUpload[side].enable := FALSE;
				WebServiceUpload[side]();
				FCreate.enable	:= FALSE;
				FCreate();
			END_IF
		//**********************************************************************************************
		// Upload file
		//**********************************************************************************************
		EXP_FILE_UPLOAD_2:
			// Show current state
			animation := WorkingStatus(ADR(EXPL), ADR('upload - saving file...'), animation);

			// ----------------------------------------------------------------------------------------
			// Initialize file write structure
			FWrite.enable	:= TRUE;
			FWrite.ident	:= FCreate.ident;
			FWrite.len		:= file_data_len;
			FWrite.pSrc		:= AsMemPartAllocClear_0.mem + file_data_start;
			FWrite();

			// ----------------------------------------------------------------------------------------
			// OK
			IF (FWrite.status = OK) THEN
				step := EXP_FILE_UPLOAD_3;
			// Error
			ELSIF (FWrite.status <> ERR_FUB_BUSY) THEN
				step := CreateError(FWrite.status, side, step, 'error writing file from upload', ADR(EXPL));
			END_IF
		//**********************************************************************************************
		// Upload file
		//**********************************************************************************************
		EXP_FILE_UPLOAD_3:
			// ----------------------------------------------------------------------------------------
			// Initialize file close structure
			FClose.enable	:= TRUE;
			FClose.ident	:= FCreate.ident;
			FClose();

			// ----------------------------------------------------------------------------------------
			// OK
			IF (FClose.status = OK) THEN
				brsmemset(AsMemPartAllocClear_0.mem, 0, EXPL_UPLOAD_DOWNLOAD_SIZE);
				WebServiceUpload[side].enable := FALSE;
				WebServiceUpload[side]();
				EXPL.CMD[side].upload := FALSE;
				EXPL.VIS[side].reload_upload := TRUE;
				// Report error from file write
				IF (FWrite.status <> ERR_OK) THEN
					step := CreateError(FWrite.status, side, step, 'error writing file from upload', ADR(EXPL));
				ELSE
					EXPL.CMD[side].refresh := 1;
					step := EXP_WAIT;
				END_IF
			// Error
			ELSIF (FClose.status <> ERR_FUB_BUSY) THEN
				step := CreateError(FClose.status, side, step, 'error closing file from upload', ADR(EXPL));
			END_IF
		//**********************************************************************************************
		// Create new directory
		//**********************************************************************************************
		EXP_DIR_CREATE:
			// Show current state
			animation := WorkingStatus(ADR(EXPL), ADR('creating directory...'), animation);

			// ----------------------------------------------------------------------------------------
			// Initialize directory create structure
			CreateCompletePath(EXPL.PAR[side].dir_path, EXPL.PAR[side].new_name, ADR(tmp_str3));
			DCreate.enable	:= 1;
			DCreate.pDevice := ADR(EXPL.PAR[side].device_active);
			DCreate.pName 	:= ADR(tmp_str3);
			DCreate();

			// ----------------------------------------------------------------------------------------
			// OK
			IF (DCreate.status = OK) THEN
				// Reset command and return to wait state
				EXPL.CMD[side].dir_create 	:= FALSE;
				EXPL.CMD[side].refresh 		:= TRUE;
				step := EXP_WAIT;
			// Error
			ELSIF (DCreate.status <> ERR_FUB_BUSY) THEN
				step := CreateError(DCreate.status, side, step, 'error creating directory', ADR(EXPL));
			END_IF
		//**********************************************************************************************
		// Delete selected directory
		//**********************************************************************************************
		EXP_DIR_DELETE:
			// Show current state
			animation := WorkingStatus(ADR(EXPL), ADR('deleting directory...'), animation);

			// ----------------------------------------------------------------------------------------
			// Initialize directory delete structure
			CreateCompletePath(EXPL.PAR[side].dir_path, item_name, ADR(tmp_str3));
			DDelete.enable	:= TRUE;
			DDelete.pDevice := ADR(EXPL.PAR[side].device_active);
			DDelete.pName 	:= ADR(tmp_str3);
			DDelete();

			// ----------------------------------------------------------------------------------------
			// OK
			IF (DDelete.status = OK) THEN
				// Reset command and return to wait state
				EXPL.CMD[side].delete := FALSE;
				EXPL.CMD[side].refresh := TRUE;
				step := EXP_WAIT;
			// Error
			ELSIF (DDelete.status <> ERR_FUB_BUSY) THEN
				step := CreateError(DDelete.status, side, step, 'error deleting directory', ADR(EXPL));
			END_IF
		//**********************************************************************************************
		// Rename selected directory
		//**********************************************************************************************
		EXP_DIR_RENAME:
			// Show current state
			animation := WorkingStatus(ADR(EXPL), ADR('renaming directory...'), animation);

			// ----------------------------------------------------------------------------------------
			// Initialize file delete structure
			CreateCompletePath(EXPL.PAR[side].dir_path, EXPL.DAT[side].item_list[EXPL.VIS[side].item_selected], ADR(tmp_str2));
			CreateCompletePath(EXPL.PAR[side].dir_path, EXPL.PAR[side].new_name, ADR(tmp_str3));
			DRename.enable		:= TRUE;
			DRename.pDevice 	:= ADR(EXPL.PAR[side].device_active);
			DRename.pName		:= ADR(tmp_str2);
			DRename.pNewName	:= ADR(tmp_str3);
			DRename();

			// ----------------------------------------------------------------------------------------
			// OK
			IF (DRename.status = OK) THEN
				// Reset command and return to wait state
				EXPL.CMD[side].rename 	:= FALSE;
				EXPL.CMD[side].refresh  := TRUE;
				step := EXP_WAIT;
				// Error
			ELSIF (DRename.status <> ERR_FUB_BUSY) THEN
				step := CreateError(DRename.status, side, step, 'error renaming directory', ADR(EXPL));
			END_IF
		//**********************************************************************************************
		// Overwrite file - Check if file exists
		//**********************************************************************************************
		EXP_OVERWRITE_1:
			// ----------------------------------------------------------------------------------------
			// Checking for files with the same name
			EXPL.VIS[side].upload_overwrite_response := 0;

			FOR lx:=0 TO EXPL.DAT[side].item_num DO
				IF((EXPL.CMD[side].copy = TRUE AND EXPL.DAT[NOT side].item_list[lx] = item_name) OR (EXPL.CMD[side].upload = TRUE AND EXPL.DAT[side].item_list[lx] = item_name)) THEN
					EXPL.VIS[side].upload_overwrite_request	:= TRUE;
					step := EXP_OVERWRITE_2;
					RETURN;
				END_IF;
			END_FOR;
			EXPL.VIS[side].upload_overwrite_response := SKIP;
			step := EXP_OVERWRITE_2;
		//**********************************************************************************************
		// Overwrite file - Wait for message box response
		//**********************************************************************************************
		EXP_OVERWRITE_2:
			// Overwrite file
			IF(EXPL.VIS[side].upload_overwrite_response = YES OR EXPL.VIS[side].upload_overwrite_response = SKIP) THEN
				// Proceed with copy command
				IF(EXPL.CMD[side].copy = TRUE) THEN
					IF(brsmemcmp(ADR(item_name), ADR('(DIR)'), 5) = 0)	THEN
						step := EXP_DIR_COPY;
					ELSE
						step := EXP_FILE_COPY;
					END_IF
				// Proceed with upload command
				ELSE
					IF(EXPL.VIS[side].upload_overwrite_response = SKIP) THEN
						step := EXP_FILE_UPLOAD_1;
					ELSE
						step := EXP_FILE_DELETE;
					END_IF
				END_IF
				EXPL.VIS[side].upload_overwrite_request	:= FALSE;
			// Do not overwrite file
			ELSIF(EXPL.VIS[side].upload_overwrite_response = NO) THEN
				// Reset upload command
				brsmemset(AsMemPartAllocClear_0.mem, 0, EXPL_UPLOAD_DOWNLOAD_SIZE);
				WebServiceUpload[side].enable := FALSE;
				WebServiceUpload[side]();
				EXPL.CMD[side].upload := FALSE;
				EXPL.VIS[side].reload_upload := TRUE;
				// Reset copy command
				EXPL.CMD[side].copy	:= FALSE;

				EXPL.VIS[side].upload_overwrite_request	:= FALSE;
				step := EXP_WAIT;
			END_IF
	END_CASE

END_PROGRAM
```

### Program Logical/mappFileExplorer/USBdevice (IEC) - Sample for all AsUSB-Library-Functions

#### USBdevice.st - Cyclic code
```iecst
PROGRAM _INIT
END_PROGRAM

PROGRAM _CYCLIC

	CASE USB.PAR.state_machine OF
		// -----------------------------------------------------------------------------------------------------------
		// Wait state
		// -----------------------------------------------------------------------------------------------------------
		USB_WAIT:
			// Refresh USB data every X seconds when enabled
			IF USB.CMD.auto_scan = TRUE THEN
				TON_10ms_01(IN:=1, PT:=USB.PAR.refresh_interval);
				// Get new USB data
				IF(TON_10ms_01.Q) THEN
					TON_10ms_01(IN:=0);
					node := 0;
					brsmemset(ADR(usb_data), 0, SIZEOF(usb_data));
					USB.PAR.state_machine := USB_CREATE_NODE_ID_LIST;
				END_IF
			ELSE
				TON_10ms_01(IN:=0);
			END_IF;
			// Refresh USB data every X seconds when enabled
			IF USB.CMD.error_reset = TRUE THEN
				USB.PAR.state_machine := USB_ERROR;
			END_IF;
		// -----------------------------------------------------------------------------------------------------------
		// Get USB device list
		// -----------------------------------------------------------------------------------------------------------
		USB_CREATE_NODE_ID_LIST:
			UsbNodeListGet_0.enable := 1;
			UsbNodeListGet_0.pBuffer := ADR(node_id_buffer);
			UsbNodeListGet_0.bufferSize := SIZEOF(node_id_buffer);
			UsbNodeListGet_0.filterInterfaceClass := asusb_CLASS_MASS_STORAGE;
			UsbNodeListGet_0.filterInterfaceSubClass := 0;
			UsbNodeListGet_0;

			// --------------------------------------------------------------------------------------------------------------------
			// Success
			IF UsbNodeListGet_0.status = 0 THEN
				USB.PAR.state_machine := USB_READ_DEVICE_DATA;
				// No USB devices found
			ELSIF UsbNodeListGet_0.status = asusbERR_USB_NOTFOUND THEN
				// Unlink old device if it is gone now otherwise wait for next round
				IF(USB.PAR.is_connected) THEN
					USB.PAR.state_machine := USB_UNLINK_DEVICE;
				ELSE
					USB.PAR.state_machine := USB_WAIT;
				END_IF
				// Error
			ELSIF UsbNodeListGet_0.status <> ERR_FUB_BUSY THEN
				USB.ERR.state := USB.PAR.state_machine;
				USB.ERR.text := 'error getting device list';
				USB.PAR.state_machine := USB_ERROR;
			END_IF;
		// -----------------------------------------------------------------------------------------------------------
		// Get device information
		// -----------------------------------------------------------------------------------------------------------
		USB_READ_DEVICE_DATA:
			UsbNodeGet_0.enable := 1;
			UsbNodeGet_0.nodeId := node_id_buffer[node];
			UsbNodeGet_0.pBuffer := ADR(usb_data[node]);
			UsbNodeGet_0.bufferSize := SIZEOF (usb_data[node]);
			UsbNodeGet_0;

			// --------------------------------------------------------------------------------------------------------------------
			// Success
			IF UsbNodeGet_0.status = 0 THEN
				// Make sure we have enough space to store USB data, proceed with next USB.PAR.state_machine when all devices are detetced
				IF (node = UsbNodeListGet_0.listNodes - 1) OR (node > SIZEOF(usb_data)/SIZEOF(usb_data[0])) THEN
					idx := 0;
					USB.PAR.state_machine := USB_CHECK_DEVICE;
					// Get next USB device
				ELSE
					node := node + 1;
				END_IF;
				// Error
			ELSIF UsbNodeGet_0.status <> ERR_FUB_BUSY THEN
				USB.ERR.state := USB.PAR.state_machine;
				USB.ERR.text := 'error getting device data';
				USB.PAR.state_machine := USB_ERROR;
			END_IF;
		// -----------------------------------------------------------------------------------------------------------
		// Check if device is connected
		// -----------------------------------------------------------------------------------------------------------
		USB_CHECK_DEVICE:
			// Check if device is already linked
			IF(USB.PAR.is_connected) THEN
				// Device is already linked, return to wait state
				IF(brsmemcmp(ADR(usb_data_linked), ADR(usb_data[idx]), SIZEOF(usb_data[idx])) = 0) THEN
					USB.PAR.state_machine := USB_WAIT;
					// Check next device
				ELSIF(idx < node) THEN
					idx := idx + 1;
					// Unlink device if it is gone
				ELSE
					USB.PAR.state_machine := USB_UNLINK_DEVICE;
				END_IF
			ELSE
				// Check if B&R dongle should be excluded from list
				IF(USB.PAR.ignore_dongle=TRUE AND usb_data[idx].productId=1001 AND usb_data[idx].vendorId=1615) THEN
					IF(idx < node) THEN
						idx := idx + 1;
					ELSE
						USB.PAR.state_machine := USB_WAIT;
					END_IF
				ELSE
					USB.PAR.state_machine := USB_LINK_DEVICE;
				END_IF
			END_IF
		// -----------------------------------------------------------------------------------------------------------
		// Link device
		// -----------------------------------------------------------------------------------------------------------
		USB_LINK_DEVICE:
			// Create device string
			brsstrcpy(ADR(device_param), ADR('/DEVICE='));
			brsstrcat(ADR(device_param), ADR(usb_data[node].ifName));
			// Link device
			DevLink_0.enable := 1;
			DevLink_0.pDevice := ADR('USB_DEVICE');
			DevLink_0.pParam := ADR(device_param);
			DevLink_0;

			// --------------------------------------------------------------------------------------------------------------------
			// Success
			IF DevLink_0.status = 0 THEN
				brsmemcpy(ADR(usb_data_linked), ADR(usb_data[node]), SIZEOF(usb_data[node]));
				USB.PAR.is_connected := TRUE;
				USB.PAR.state_machine := USB_WAIT;
				// Error
			ELSIF DevLink_0.status <> ERR_FUB_BUSY THEN
				USB.ERR.state := USB.PAR.state_machine;
				USB.ERR.text := 'error linking device';
				USB.PAR.state_machine := USB_ERROR;
			END_IF;
		// -----------------------------------------------------------------------------------------------------------
		// UnLink device
		// -----------------------------------------------------------------------------------------------------------
		USB_UNLINK_DEVICE:
			DevUnlink_0.enable := 1;
			DevUnlink_0.handle := DevLink_0.handle;
			DevUnlink_0;

			// --------------------------------------------------------------------------------------------------------------------
			// Success
			IF DevUnlink_0.status = 0 THEN
				brsmemset(ADR(usb_data_linked), 0, SIZEOF(usb_data_linked));
				USB.PAR.is_connected := FALSE;
				IF(UsbNodeListGet_0.status = asusbERR_USB_NOTFOUND) THEN
					USB.PAR.state_machine := USB_WAIT;
				ELSE
					idx := 0;
					USB.PAR.state_machine := USB_CHECK_DEVICE;
				END_IF
				// Error
			ELSIF DevUnlink_0.status <> ERR_FUB_BUSY THEN
				USB.ERR.state := USB.PAR.state_machine;
				USB.ERR.text := 'error unlinking device';
				USB.PAR.state_machine := USB_ERROR;
			END_IF;
		// -----------------------------------------------------------------------------------------------------------
		// Error state
		// -----------------------------------------------------------------------------------------------------------
		USB_ERROR:
			// Get more error information
			USB.ERR.no := FileIoGetSysError();
			USB.ERR.active := TRUE;
			USB.PAR.is_connected := FALSE;

			// Unlink device
			DevUnlink_0.enable := 1;
			DevUnlink_0.handle := DevLink_0.handle;
			DevUnlink_0;

			// Reset error
			IF(USB.CMD.error_reset AND DevUnlink_0.status <> ERR_FUB_BUSY) THEN
				USB.CMD.error_reset := FALSE;
				USB.ERR.active := FALSE;
				USB.ERR.no := 0;
				brsmemset(ADR(USB.ERR.text), 0, SIZEOF(USB.ERR.text));
				USB.PAR.state_machine := USB_WAIT;
			END_IF
	END_CASE;

END_PROGRAM

PROGRAM _EXIT
	REPEAT
		DevUnlink_0.enable := 1;
		DevUnlink_0.handle := DevLink_0.handle;
		DevUnlink_0;
		UNTIL DevUnlink_0.status <> ERR_FUB_BUSY
	END_REPEAT;
END_PROGRAM
```

#### USBdevice.var - Data for read_data Task
```iecst
(*----------------------------------------------------------------------------------------------------------------------------------------------------------------------------------------------------------------------------------------------------------------------*)
(*Local constants*)
VAR CONSTANT
	WAIT : USINT := 0; (*Function step: Wait for starting the Function chain*)
	CREATE_NODE_ID_LIST : USINT := 1; (*Function step: Create a list of Node-IDs from all active USB devices*)
	READ_DEVICE_DATA : USINT := 2; (*Function step: Read out the specific data from the Node-IDs*)
	CHECK_DEVICE : USINT := 3; (*Function step: Check file device data*)
	LINK_DEVICE : USINT := 4; (*Function step: Link file device*)
	UNLINK_DEVICE : USINT := 5; (*Function step: Unlink the File Device from specific path*)
	ERROR : USINT := 6; (*Function step: Jump to this step in every case of Error occuring in the Function chain*)
END_VAR
(*----------------------------------------------------------------------------------------------------------------------------------------------------------------------------------------------------------------------------------------------------------------------*)
(*Local functions*)
VAR
	TON_10ms_01 : TON_10ms;
	UsbNodeListGet_0 : UsbNodeListGet; (*Type of FUB UsbNodeListGet*)
	UsbNodeGet_0 : UsbNodeGet; (*Type of FUB UsbNodeGet*)
	DevLink_0 : DevLink; (*Type of FUB DevLink*)
	DevUnlink_0 : DevUnlink; (*Type of FUB DevUnlink*)
END_VAR
(*----------------------------------------------------------------------------------------------------------------------------------------------------------------------------------------------------------------------------------------------------------------------*)
(*Local variables*)
VAR
	device_param : STRING[80]; (*Connection path of USB device*)
	usb_data : ARRAY[0..4] OF usbNode_typ; (*Data of all available USB devices*)
	usb_data_linked : usbNode_typ; (*Data of the linked device*)
	node_id_buffer : ARRAY[0..4] OF UDINT; (*Different nodeIDs saved in array-elements*)
	node : USINT; (*Node number*)
	idx : USINT;
END_VAR
```

### Program Logical/mappFileExplorer/NETdevice (IEC)

#### Main.st - Init, cyclic, exit code
```iecst
PROGRAM _INIT
	(* Insert code here *)

END_PROGRAM

PROGRAM _CYCLIC

	CASE NET.PAR.state_machine OF
		// -----------------------------------------------------------------------------------------------------------
		// Wait state
		// -----------------------------------------------------------------------------------------------------------
		NET_WAIT:
			NET.PAR.enable_connect := TRUE;
			// --------------------------------------------------------------------------------------------------------------------
			// Connect to server
			IF(NET.CMD.connect) THEN
				IF(NET.PAR.is_linked) THEN
					DevUnlink_0.enable := 0;
					DevUnlink_0;
					IF (DevUnlink_0.status = ERR_FUB_ENABLE_FALSE) THEN
						NET.PAR.state_machine := NET_UNLINK_DEVICE;
					END_IF
				ELSE
					DevLink_0.enable := 0;
					DevLink_0;
					IF (DevLink_0.status = ERR_FUB_ENABLE_FALSE) THEN
						NET.PAR.state_machine := NET_LINK_DEVICE;
					END_IF
				END_IF
			END_IF
			// --------------------------------------------------------------------------------------------------------------------
			// Disconnect from server
			IF(NET.CMD.error_reset) THEN
				IF(NET.PAR.is_linked) THEN
					DevUnlink_0.enable := 0;
					DevUnlink_0;
					NET.PAR.state_machine := NET_UNLINK_DEVICE;
				ELSE
					NET.CMD.error_reset := FALSE;
				END_IF
			END_IF
		// -----------------------------------------------------------------------------------------------------------
		// Link device
		// -----------------------------------------------------------------------------------------------------------
		NET_LINK_DEVICE:
			// Create device string
			NET.PAR.enable_connect := FALSE;
			brsmemset(ADR(device_param), 0, SIZEOF(device_param));
			IF(brsstrcmp(ADR(NET.PAR.server_name), ADR('')) <> 0) THEN
				brsstrcat(ADR(device_param), ADR('/SNAME='));
				brsstrcat(ADR(device_param), ADR(NET.PAR.server_name));
				brsstrcat(ADR(device_param), ADR(' '));
			END_IF
			IF(brsstrcmp(ADR(NET.PAR.server_ip), ADR('')) <> 0) THEN
				brsstrcat(ADR(device_param), ADR('/SIP='));
				brsstrcat(ADR(device_param), ADR(NET.PAR.server_ip));
				brsstrcat(ADR(device_param), ADR(' '));
			END_IF
			IF(brsstrcmp(ADR(NET.PAR.server_protocol), ADR('')) <> 0) THEN
				brsstrcat(ADR(device_param), ADR('/PROTOCOL='));
				brsstrcat(ADR(device_param), ADR(NET.PAR.server_protocol));
				brsstrcat(ADR(device_param), ADR(' '));
			END_IF
			IF(brsstrcmp(ADR(NET.PAR.server_port), ADR('')) <> 0) THEN
				brsstrcat(ADR(device_param), ADR('/PORT='));
				brsstrcat(ADR(device_param), ADR(NET.PAR.server_port));
				brsstrcat(ADR(device_param), ADR(' '));
			END_IF
			IF(brsstrcmp(ADR(NET.PAR.server_domain), ADR('')) <> 0) THEN
				brsstrcat(ADR(device_param), ADR('/DOMAIN='));
				brsstrcat(ADR(device_param), ADR(NET.PAR.server_domain));
				brsstrcat(ADR(device_param), ADR(' '));
			END_IF
			IF(brsstrcmp(ADR(NET.PAR.server_share), ADR('')) <> 0) THEN
				brsstrcat(ADR(device_param), ADR('/SHARE='));
				brsstrcat(ADR(device_param), ADR(NET.PAR.server_share));
				brsstrcat(ADR(device_param), ADR(' '));
			END_IF
			IF(brsstrcmp(ADR(NET.PAR.user_name), ADR('')) <> 0) THEN
				brsstrcat(ADR(device_param), ADR('/USER='));
				brsstrcat(ADR(device_param), ADR(NET.PAR.user_name));
				brsstrcat(ADR(device_param), ADR(' '));
			END_IF
			IF(brsstrcmp(ADR(NET.PAR.user_password), ADR('')) <> 0) THEN
				brsstrcat(ADR(device_param), ADR('/PASSWORD='));
				brsstrcat(ADR(device_param), ADR(NET.PAR.user_password));
				brsstrcat(ADR(device_param), ADR(' '));
			END_IF

			// Link device
			DevLink_0.enable := 1;
			DevLink_0.pDevice := ADR('NET_DEVICE');
			DevLink_0.pParam := ADR(device_param);
			DevLink_0;

			// --------------------------------------------------------------------------------------------------------------------
			// Success
			IF DevLink_0.status = 0 THEN
				device_handle := DevLink_0.handle;
				NET.PAR.is_linked := TRUE;
				NET.CMD.connect := FALSE;
				NET.PAR.state_machine := NET_WAIT;
			// --------------------------------------------------------------------------------------------------------------------
			// Abort command
			ELSIF(NET.CMD.error_reset) THEN
				NET.CMD.error_reset := FALSE;
				NET.CMD.connect := FALSE;
				NET.PAR.state_machine := NET_WAIT;
				// Error
			ELSIF DevLink_0.status <> ERR_FUB_BUSY THEN
				NET.ERR.state := NET.PAR.state_machine;
				NET.ERR.no := DevLink_0.status;
				NET.ERR.text := 'error linking device';
				NET.PAR.state_machine := NET_ERROR;
			END_IF;
		// -----------------------------------------------------------------------------------------------------------
		// UnLink device
		// -----------------------------------------------------------------------------------------------------------
		NET_UNLINK_DEVICE:
			NET.PAR.enable_connect := FALSE;
			DevUnlink_0.enable := 1;
			DevUnlink_0.handle := device_handle;
			DevUnlink_0;

			// --------------------------------------------------------------------------------------------------------------------
			// Success
			IF DevUnlink_0.status = 0 THEN
				NET.PAR.is_linked := FALSE;
				IF(NET.CMD.connect) THEN
					DevLink_0.enable := 0;
					DevLink_0;
					NET.PAR.state_machine := NET_LINK_DEVICE;
				ELSE
					NET.CMD.error_reset := FALSE;
					NET.PAR.state_machine := NET_WAIT;
				END_IF
			// Error
			ELSIF DevUnlink_0.status <> ERR_FUB_BUSY THEN
				NET.CMD.error_reset := FALSE;
				NET.ERR.state := NET.PAR.state_machine;
				NET.ERR.no := DevUnlink_0.status;
				NET.ERR.text := 'error unlinking device';
				NET.PAR.state_machine := NET_ERROR;
			END_IF;
		// -----------------------------------------------------------------------------------------------------------
		// Error step
		// -----------------------------------------------------------------------------------------------------------
		NET_ERROR:
			// Reset commands
			NET.PAR.enable_connect := FALSE;
			NET.CMD.connect := FALSE;

			// Get more error information
			IF(NET.ERR.no = 0) THEN
				NET.ERR.no := FileIoGetSysError();
			END_IF
			NET.ERR.active := TRUE;
			IF(NET.ERR.no=26228) THEN
				brsstrcpy(ADR(NET.ERR.text), ADR('connection rejected: check network protocol, username and password'));
			ELSIF(DevLink_0.status = fiERR_DEVICE_ALREADY_EXIST) THEN
				brsstrcpy(ADR(NET.ERR.text), ADR('device is already connected'));
			END_IF

			// Reset error
			IF(NET.CMD.error_reset) THEN
				NET.CMD.error_reset := FALSE;
				NET.ERR.active := FALSE;
				NET.ERR.no := 0;
				brsmemset(ADR(NET.ERR.text), 0, SIZEOF(NET.ERR.text));
				NET.PAR.state_machine := NET_WAIT;
			END_IF
	END_CASE;

END_PROGRAM

PROGRAM _EXIT
	REPEAT
		DevUnlink_0.enable := 1;
		DevUnlink_0.handle := DevLink_0.handle;
		DevUnlink_0;
		UNTIL DevUnlink_0.status <> ERR_FUB_BUSY
	END_REPEAT;
END_PROGRAM
```

#### Variables.var - Local variables
```iecst
(*----------------------------------------------------------------------------------------------------------------------------------------------------------------------------------------------------------------------------------------------------------------------*)
(*Local constants*)
VAR CONSTANT
	WAIT : USINT := 0; (*Function step: Wait for starting the Function chain*)
	LINK_DEVICE : USINT := 1; (*Function step: Link file device*)
	UNLINK_DEVICE : USINT := 2; (*Function step: Unlink the File Device from specific path*)
	ERROR : USINT := 3; (*Function step: Jump to this step in every case of Error occuring in the Function chain*)
END_VAR
(*----------------------------------------------------------------------------------------------------------------------------------------------------------------------------------------------------------------------------------------------------------------------*)
(*Local functions*)
VAR
	DevLink_0 : DevLink; (*Type of FUB DevLink*)
	DevUnlink_0 : DevUnlink; (*Type of FUB DevUnlink*)
END_VAR
(*----------------------------------------------------------------------------------------------------------------------------------------------------------------------------------------------------------------------------------------------------------------------*)
(*Local variables*)
VAR
	device_param : STRING[200]; (*Connection path of USB device*)
	device_handle : UDINT;
END_VAR
```

### changelog.txt
```
Version 1.3
- Code cleanup
- Added file device memory information
- Change from static IP to DHCP
- Fixed filter text field and button is disabled when no files are visible
- Fixed file size calculation
- Fixed ReplaceString function call

Version 1.2
- Fixed download not working when downloading the same file again
- Fixed upload not working with large files > 1 MB

Version 1.1
- Fixed file open click event
- Added support multiple USB sticks
- Added message box when uploading or copying file that exists on target
- Fixed button rename is not disabled when command is running

Version 1.0
- Added support for file download over mappView
- Added support for file upload over mappView
- Code cleanup

Version 0.9
- Added function to view files by double click or command

Version 0.8
- Added function for generating list box data provider
- Fixed typos, cleaned up binding file
- Created individual packages for NET and USB
- Fixed enable/disable
- Added message box before deleting an item

Version 0.7
- New function rename file or folder
- Fixed memory leak when last entry in list is used
- Code optimizations

Version 0.6
- Changed upper limit of USB polling interval
- Removed obsolete error numbers
- Replaced error numbers with constants
- Removed obsolete variables
- Fixed old_filter variable size
- Fixed file size added to file name
- Disable file device and filter during operation

Version 0.5
- Main task ported to structure text
- Allow oversized names for files and folders
- Fixed variables types
- Applied python naming convention to all code

Version 0.2
- Added configuration for network connections
- Code cleanup

Version 0.1
- First public release
```

### PackageTypes.typ - not listed in the package file held
```iecst
TYPE
	ClientInfoType : 	STRUCT
		userId : WSTRING[80];
		isValid : BOOL;
		ipAddress : WSTRING[15];
		languageId : WSTRING[2];
		screenResolution : WSTRING[32];
		slotId : SINT;
	END_STRUCT;
	typERR_EXP : 	STRUCT
		txt : STRING[100]; (* Error text *)
		nr : UINT; (* Error number *)
		step : USINT; (* Error step *)
	END_STRUCT;
	typCMD_EXP : 	STRUCT
		refresh : BOOL; (* Read directory and file names from devices *)
		dir_change : BOOL; (* Change current directory *)
		dir_create : BOOL; (* Create a new directory *)
		copy : BOOL; (* Copy selected item from device a TO device b *)
		copyall : BOOL; (* Copy all items from device a TO device b	*)
		delete : BOOL; (* Delete selected file *)
	END_STRUCT;
	typPAR_EXP : 	STRUCT
		device_active : STRING[40]; (* Device name *)
		device_list : ARRAY[0..4]OF STRING[40]; (* Device name *)
		item_filter : STRING[4]; (* Only show files with this extension	*)
		dir_name : STRING[DIR_PATH_SIZE]; (* Directory name for create *)
		dir_path : STRING[DIR_PATH_SIZE]; (* Current directory path	*)
	END_STRUCT;
	typDAT_EXP : 	STRUCT
		item_list : ARRAY[0..DAT_LIST_NUM]OF STRING[DAT_ITEM_SIZE]; (* List with file names	*)
		item_size : ARRAY[0..DAT_LIST_NUM]OF STRING[DAT_SIZE_SIZE]; (* List with file names *)
		item_num : UINT; (* Number OF files	*)
	END_STRUCT;
	typVIS_EXP : 	STRUCT
		item_selected : UINT; (* Current selected file *)
		enable_copy_delete : BOOL; (*Enable or disable buttons copy and delete*)
		double_click_dir_change : USINT;
		device_list : ARRAY[0..4]OF STRING[80]; (* Device name *)
	END_STRUCT;
	typMain_EXP : 	STRUCT
		CMD : ARRAY[0..1]OF typCMD_EXP; (* Command structure *)
		PAR : ARRAY[0..1]OF typPAR_EXP; (* Parameter structure *)
		DAT : ARRAY[0..1]OF typDAT_EXP;
		VIS : ARRAY[0..1]OF typVIS_EXP;
		ERR : typERR_EXP; (* Error structure *)
		status : STRING[50]; (* Actual step	*)
	END_STRUCT;
END_TYPE
```

### PackageVariables.var - not listed in the package file held
```iecst
VAR CONSTANT
	DIR_PATH_SIZE : UINT := 200; (* Directory path name size							*)
	DAT_LIST_NUM : UINT := 50;
	DAT_ITEM_SIZE : USINT := 30; (* Record name size									*)
	DAT_SIZE_SIZE : USINT := 30; (* Record name size									*)
	DEVICE_LIST : ARRAY[0..4] OF STRING[40] := ['USER','SYSTEM',3('')];
END_VAR
VAR
	EXPL : typMain_EXP;
	ClientInfoCurrent : ClientInfoType;
	ClientInfo : ARRAY[0..4] OF ClientInfoType;
END_VAR
```

### UsbTypes.typ
```iecst
TYPE
	usbSTATE :
		(
		USB_WAIT, (*Wait for starting the Function chain*)
		USB_CREATE_NODE_ID_LIST, (*Create a list of Node-IDs from all active USB devices*)
		USB_READ_DEVICE_DATA, (*Read out the specific data from the Node-IDs*)
		USB_CHECK_LINKED, (*Check if device is still connected*)
		USB_LINK_NEW,
		USB_LINK_DEVICE, (*Link file device*)
		USB_UNLINK_DEVICE, (*Unlink the File Device from specific path*)
		USB_ERROR (*Jump to this step in every case of Error occuring in the Function chain*)
		);
	usbCMD : 	STRUCT
		auto_scan : BOOL := TRUE; (*Scan USB ports automatically*)
		error_reset : BOOL; (*Reset error*)
	END_STRUCT;
	usbPAR : 	STRUCT
		ignore_dongle : BOOL := TRUE; (*Ignoe B&R license dongle*)
		refresh_interval : UINT := 300; (*Intervall timer for USB device refresh*)
		is_connected : ARRAY[1..USB_MAX_CNT]OF BOOL; (*Shows if a USB stick is connected*)
	END_STRUCT;
	usbERR : 	STRUCT
		state : usbSTATE; (*State where the error occured*)
		text : STRING[80]; (*Error text*)
	END_STRUCT;
	usbMAIN : 	STRUCT
		CMD : usbCMD; (*Command structure*)
		PAR : usbPAR; (*Parameter structure*)
		ERR : usbERR; (*Error structure*)
		status : UINT; (*Current status*)
	END_STRUCT;
END_TYPE
```

### UsbVariables.var
```iecst
VAR
	USB : usbMAIN;
END_VAR
VAR CONSTANT
	USB_MAX_CNT : USINT := 5; (*Maximum number of keys that are supported*)
END_VAR
```

### Program Logical/USBdevice/UsbDevice (IEC) - Sample for all AsUSB-Library-Functions
